// TIA Portal V16 export
// export: Created 2023-03-29T11:04:28.582078Z, ExportSetting WithDefaults, DisplayName Totally Integrated Automation Portal, DisplayVersion V16 Update 6, DisplayName TIA Portal Version Control Interface, DisplayVersion V16 Update 2, DisplayName TIA Portal Openness, DisplayVersion V16 Update 6, DisplayName STEP 7 Professional, DisplayVersion V16 Update 6, DisplayName STEP 7 Safety, DisplayVersion V16, DisplayName WinCC Advanced, DisplayVersion V16 Update 6
FUNCTION "DRV01" : Void   // FC1, LAD
TITLE = Funkcja sterowania stycznikiem silnika
{ S7_Optimized_Access := 'FALSE' }
VERSION : 0.1
// Funkcja standardowa sluzy do zalaczania silnika.
// Posiada trzy tryby pracy:
//      - localny (zalaczanie  elektrycznie bez PLC)
//      - zdalny  (zalaczanie przez PLC)
//          - reczny (zalaczanie przez dyspozytora z SCADA)
//          - automatyczny (zalaczanie wynikle z algotytmu sterowania)
// Zrodlo danych dla funkcji stanowia:
//      - sygnaly I/O PLC
//          - =REDY -gotowosc napedu
//          - =REMT -sterowanie napedu 1-zdalnie 0-local
//          - =RUN  -naped wlaczony
//          - =CB   -zalaczenie stycznika
//       - =STAT bajt statusu napedu 
//               jego kopia w DB =WIZ stanowi interface PLC/MMI
//          - bit 0 Alarm              (sygnal do MMI)
//          - bit 1  
//          - bit 2 kopia sygnalu REMT (sygnal do SCADA)
//          - bit 3 kopia sygnalu RUN  (sygnal do SCADA)
//          - bit 4 wylaczenie reczne  (sygnal z SCADA) 
//          - bit 5 wlaczenie reczne   (sygnal z SCADA)
//          - bit 6 alarm reset        (sygnal z SCADA)
//          - bit 7 1=auto, 0=man      (sygnal z SCADA)
//        - =SUPV - sygnal zalacznia w trybie automatycznym
//        - sygnaly czasowe
//          - =TMR1 -kontrola czasu zalaczenia stycznika
//          - =KT1  -wartosc czasu timera 1
//          - flagi
// stored: AutoNumber false, IsIECCheckEnabled false, SetENOAutomatically false, UDAEnableTagReadback false
   VAR_INPUT
      REDY : Bool;   // Sygnał gotowości
      RUN : Bool;   // Sygnał pracy
      REMT : Bool;   // Sterowanie napędu zdalne-1 lokalne -0
      SUPV : Bool;   // Sygnalizacja załączenia w trybie automatycznym
      KT1 : Time;   // wartosc czasu timera 1
   END_VAR
   VAR_IN_OUT
      WIZ : Byte;   // Wektor stanu ze SCADA
      CB : Bool;   // Przekaźnik urządzenia
      TMR1 : TON_TIME;   // Kontrola czasu załączenia stycznika
      STAT : Byte;   // Wektor stanu urządzenia
   END_VAR
   // Ret_Val : Napęd jednokierunkowy - pompy
BEGIN

REGION Network 1: Network 1: mapowanie wektora statusu napędu i stanu wektora z SCADA
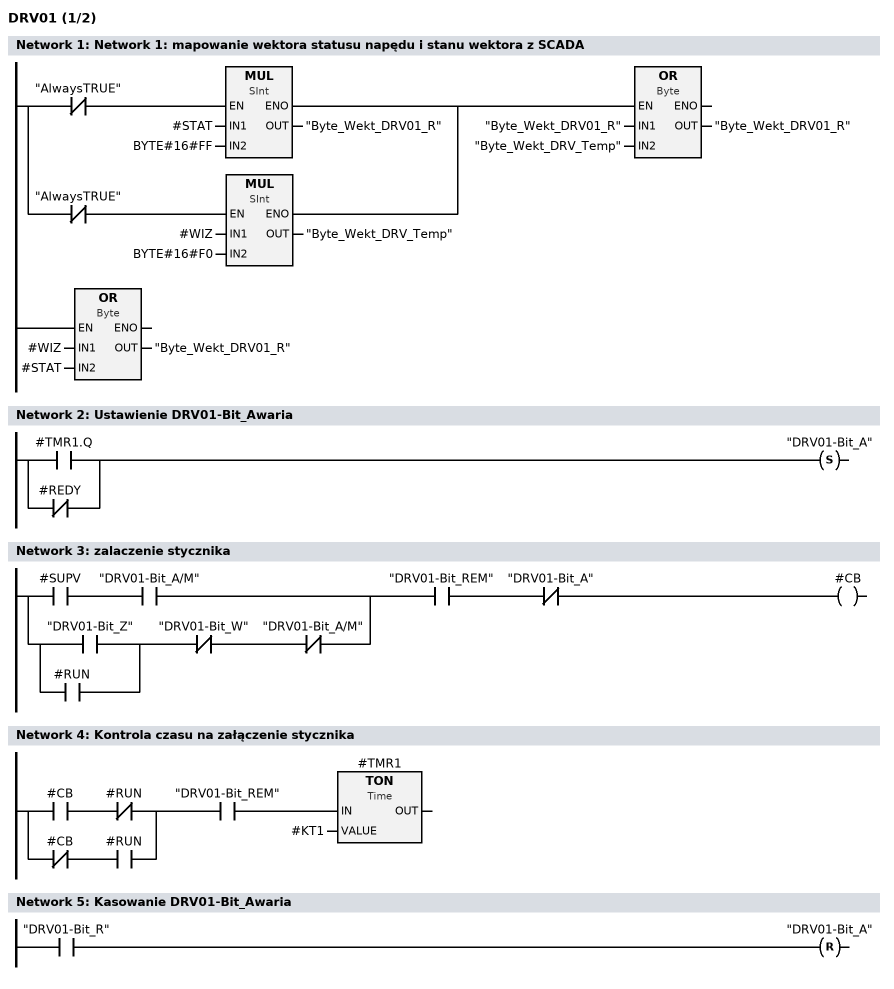
   // ENO of a box is taken as its EN; it also drops when the box reports an error
   IF NOT "AlwaysTRUE" THEN
       "Byte_Wekt_DRV01_R" := #STAT * BYTE#16#FF;
       "Byte_Wekt_DRV_Temp" := #WIZ * BYTE#16#F0;
   END_IF;
   IF NOT "AlwaysTRUE" OR NOT "AlwaysTRUE" THEN
       "Byte_Wekt_DRV01_R" := "Byte_Wekt_DRV01_R" OR "Byte_Wekt_DRV_Temp";
   END_IF;
   "Byte_Wekt_DRV01_R" := #WIZ OR #STAT;
END_REGION

REGION Network 2: Ustawienie DRV01-Bit_Awaria
   RUNG wire#powerrail
      Contact( #TMR1.Q )
      wire#w1
      S_Coil( "DRV01-Bit_A" )
   END_RUNG
   RUNG wire#powerrail
      I_Contact( #REDY )
   END_RUNG wire#w1
   // the same network as SCL:
   IF #TMR1.Q OR NOT #REDY THEN "DRV01-Bit_A" := TRUE; END_IF;
END_REGION

REGION Network 3: zalaczenie stycznika
   RUNG wire#powerrail
      Contact( #SUPV )
      Contact( "DRV01-Bit_A/M" )
      wire#w1
      Contact( "DRV01-Bit_REM" )
      I_Contact( "DRV01-Bit_A" )
      Coil( #CB )
   END_RUNG
   RUNG wire#powerrail
      Contact( "DRV01-Bit_Z" )
      wire#w2
      I_Contact( "DRV01-Bit_W" )
      I_Contact( "DRV01-Bit_A/M" )
   END_RUNG wire#w1
   RUNG wire#powerrail
      Contact( #RUN )
   END_RUNG wire#w2
   // the same network as SCL:
   #CB := ((#SUPV AND "DRV01-Bit_A/M") OR (("DRV01-Bit_Z" OR #RUN) AND NOT "DRV01-Bit_W" AND NOT "DRV01-Bit_A/M")) AND "DRV01-Bit_REM" AND NOT "DRV01-Bit_A";
END_REGION

REGION Network 4: Kontrola czasu na załączenie stycznika
   #TMR1(IN := ((#CB AND NOT #RUN) OR (NOT #CB AND #RUN)) AND "DRV01-Bit_REM", PT := #KT1);   // TON coil
END_REGION

REGION Network 5: Kasowanie DRV01-Bit_Awaria
   RUNG wire#powerrail
      Contact( "DRV01-Bit_R" )
      R_Coil( "DRV01-Bit_A" )
   END_RUNG
   // the same network as SCL:
   IF "DRV01-Bit_R" THEN "DRV01-Bit_A" := FALSE; END_IF;
END_REGION

REGION Network 6: Bit Out wektora napędu sygnał Alarm
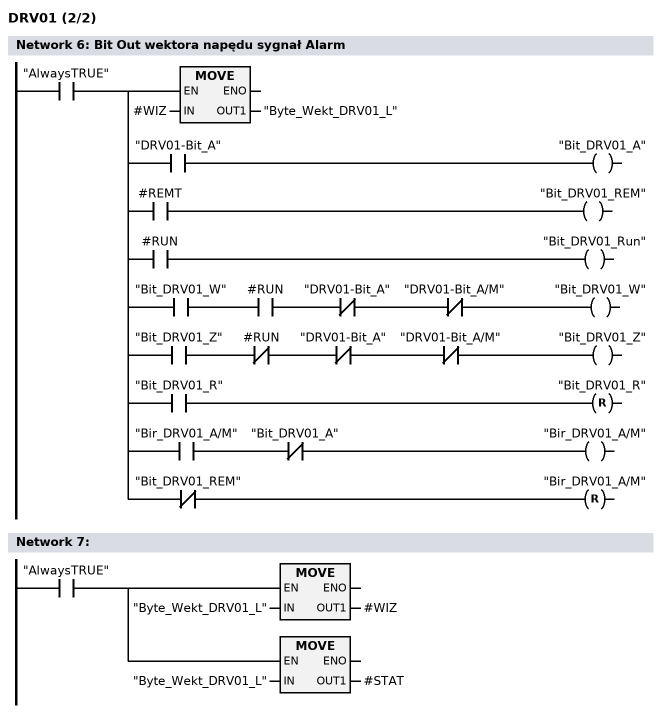
   RUNG wire#powerrail
      Contact( "AlwaysTRUE" )
      wire#w1
      { S7_GenerateENO := "TRUE" } Move(in := #WIZ, out1 => "Byte_Wekt_DRV01_L")
   END_RUNG
   RUNG wire#w1
      Contact( "DRV01-Bit_A" )
      Coil( "Bit_DRV01_A" )
   END_RUNG
   RUNG wire#w1
      Contact( #REMT )
      Coil( "Bit_DRV01_REM" )
   END_RUNG
   RUNG wire#w1
      Contact( #RUN )
      Coil( "Bit_DRV01_Run" )
   END_RUNG
   RUNG wire#w1
      Contact( "Bit_DRV01_W" )
      Contact( #RUN )
      I_Contact( "DRV01-Bit_A" )
      I_Contact( "DRV01-Bit_A/M" )
      Coil( "Bit_DRV01_W" )
   END_RUNG
   RUNG wire#w1
      Contact( "Bit_DRV01_Z" )
      I_Contact( #RUN )
      I_Contact( "DRV01-Bit_A" )
      I_Contact( "DRV01-Bit_A/M" )
      Coil( "Bit_DRV01_Z" )
   END_RUNG
   RUNG wire#w1
      Contact( "Bit_DRV01_R" )
      R_Coil( "Bit_DRV01_R" )
   END_RUNG
   RUNG wire#w1
      Contact( "Bir_DRV01_A/M" )
      I_Contact( "Bit_DRV01_A" )
      Coil( "Bir_DRV01_A/M" )
   END_RUNG
   RUNG wire#w1
      I_Contact( "Bit_DRV01_REM" )
      R_Coil( "Bir_DRV01_A/M" )
   END_RUNG
   // the same network as SCL:
   IF "AlwaysTRUE" THEN "Byte_Wekt_DRV01_L" := #WIZ; END_IF;
   "Bit_DRV01_A" := "AlwaysTRUE" AND "DRV01-Bit_A";
   "Bit_DRV01_REM" := "AlwaysTRUE" AND #REMT;
   "Bit_DRV01_Run" := "AlwaysTRUE" AND #RUN;
   "Bit_DRV01_W" := "AlwaysTRUE" AND "Bit_DRV01_W" AND #RUN AND NOT "DRV01-Bit_A" AND NOT "DRV01-Bit_A/M";
   "Bit_DRV01_Z" := "AlwaysTRUE" AND "Bit_DRV01_Z" AND NOT #RUN AND NOT "DRV01-Bit_A" AND NOT "DRV01-Bit_A/M";
   IF "AlwaysTRUE" AND "Bit_DRV01_R" THEN "Bit_DRV01_R" := FALSE; END_IF;
   "Bir_DRV01_A/M" := "AlwaysTRUE" AND "Bir_DRV01_A/M" AND NOT "Bit_DRV01_A";
   IF "AlwaysTRUE" AND NOT "Bit_DRV01_REM" THEN "Bir_DRV01_A/M" := FALSE; END_IF;
END_REGION

REGION Network 7
   RUNG wire#powerrail
      Contact( "AlwaysTRUE" )
      wire#w1
      { S7_GenerateENO := "TRUE" } Move(in := "Byte_Wekt_DRV01_L", out1 => #WIZ)
   END_RUNG
   RUNG wire#w1
      { S7_GenerateENO := "TRUE" } Move(in := "Byte_Wekt_DRV01_L", out1 => #STAT)
   END_RUNG
   // the same network as SCL:
   IF "AlwaysTRUE" THEN
       #WIZ := "Byte_Wekt_DRV01_L";
       #STAT := "Byte_Wekt_DRV01_L";
   END_IF;
END_REGION
END_FUNCTION
